// TIA Portal V16 export
// export: Created 2022-02-28T20:45:45.2571222Z, ExportSetting WithDefaults, DisplayName Totally Integrated Automation Portal, DisplayVersion V16, DisplayName TIA Portal Version Control Interface, DisplayVersion V16, DisplayName TIA Portal Openness, DisplayVersion V16, DisplayName STEP 7 Professional, DisplayVersion V16, DisplayName STEP 7 Safety, DisplayVersion V16, DisplayName WinCC Advanced, DisplayVersion V16
FUNCTION "06_Camaras" : Void   // FC6, LAD
{ S7_Optimized_Access := 'TRUE' }
VERSION : 0.1
// stored: AutoNumber true, IsIECCheckEnabled false, SetENOAutomatically false, UDAEnableTagReadback false
BEGIN

REGION Network 1: Bloque Cámara Pistilos
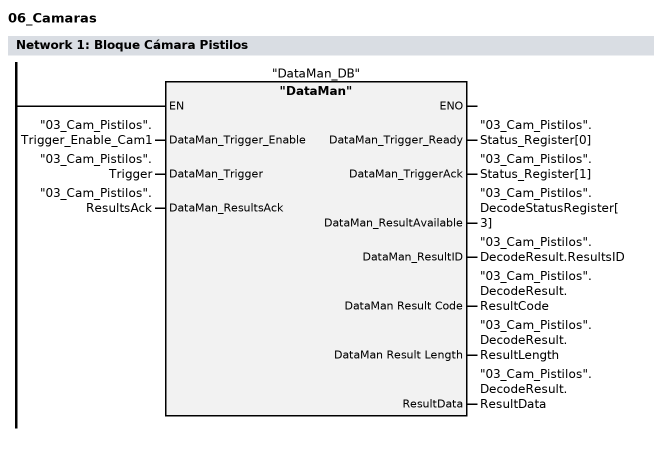
   RUNG wire#powerrail
      "DataMan_DB"(DataMan_Trigger_Enable := "03_Cam_Pistilos".Trigger_Enable_Cam1, DataMan_Trigger := "03_Cam_Pistilos".Trigger, DataMan_ResultsAck := "03_Cam_Pistilos".ResultsAck, DataMan_Trigger_Ready => "03_Cam_Pistilos".Status_Register[0], DataMan_TriggerAck => "03_Cam_Pistilos".Status_Register[1], DataMan_ResultAvailable => "03_Cam_Pistilos".DecodeStatusRegister[3], DataMan_ResultID => "03_Cam_Pistilos".DecodeResult.ResultsID, "DataMan Result Code" => "03_Cam_Pistilos".DecodeResult.ResultCode, "DataMan Result Length" => "03_Cam_Pistilos".DecodeResult.ResultLength, ResultData => "03_Cam_Pistilos".DecodeResult.ResultData)
   END_RUNG
   // the same network as SCL:
   "DataMan_DB"(DataMan_Trigger_Enable := "03_Cam_Pistilos".Trigger_Enable_Cam1,   // "DataMan"
                DataMan_Trigger := "03_Cam_Pistilos".Trigger,
                DataMan_ResultsAck := "03_Cam_Pistilos".ResultsAck,
                DataMan_Trigger_Ready => "03_Cam_Pistilos".Status_Register[0],
                DataMan_TriggerAck => "03_Cam_Pistilos".Status_Register[1],
                DataMan_ResultAvailable => "03_Cam_Pistilos".DecodeStatusRegister[3],
                DataMan_ResultID => "03_Cam_Pistilos".DecodeResult.ResultsID,
                "DataMan Result Code" => "03_Cam_Pistilos".DecodeResult.ResultCode,
                "DataMan Result Length" => "03_Cam_Pistilos".DecodeResult.ResultLength,
                ResultData => "03_Cam_Pistilos".DecodeResult.ResultData);
END_REGION
END_FUNCTION
